Staubli VAL3: action_do.pgx

program action_do(ActionItem& x_aAction[] (dimensions=1), num x_nIndex (dimensions=1))
  local num i
  local num j
  local bool l_bExit
  local num l_nClock
  local num l_nDistance
  local num l_nResult
  local string l_sData
  local string l_sEmpty
  local string l_sInstr
  local string l_sInstruction
  local string l_sType
begin
  // check if not empty...
  if x_aAction.iInstr[0].sType!="" or x_aAction.iInstr[1].sType!="" or x_aAction.iInstr[2].sType!=""
    if saveData:bDebug
      ? "ACTION INSERT,"+x_aAction.iInstr.sType+" "+x_aAction.iInstr.sData+",ID="+toString(".3",getMoveId())+","+toString(".3",clock()-cycleStatus:nTime)+",x_ID="+toString("",x_aAction.nMoveId)+",x_Dist="+toString(".2",x_aAction.nDistance)
    endIf
    l_nClock=clock()
    // wait the correct moveID
    wait((x_aAction.nMoveId+x_aAction.nDistance)<=getMoveId() or (isEmpty()) and !cycleStatus:bPause)
    // look if there are several sAction in the traj
    for i=0 to (size(x_aAction.iInstr)-1)
      // check for not empty space
      if x_aAction.iInstr[i].sType!=""
        // get the instruction
        l_sData=x_aAction.iInstr[i].sData
        l_sType=x_aAction.iInstr[i].sType
        call saveInOut:replaceIO(l_sData,l_sType,l_sData)
        l_sInstr=l_sType+" "+l_sData
        if saveData:bDebug
          ? "ACTION RUNNING,"+l_sInstr+",ID="+toString(".3",getMoveId())+","+toString(".3",clock()-cycleStatus:nTime)+",MoveID="+toString("",x_aAction.nMoveId)+",Dist="+toString(".2",x_aAction.nDistance)
        endIf
        // PRINT LOG
        if cycleStatus:bCycle
          if x_aAction.nPointId!=-1
            // is inside a trajectory
            call cycleStatus:printLog(" ."+l_sInstr)
          else
            // is outside a trajectory
            call cycleStatus:printLog("-"+l_sInstr)
          endIf
        endIf
        cycleStatus:sToShow=l_sInstr
        cycleStatus:sLastAction=l_sInstr
        if x_aAction.nPointId==-1
          // refresh the LINE of the program...
          cycleStatus:bTraj=false
          cycleStatus:nEvent=x_nIndex
        endIf
        //
        // RUN THE ACTION
        //
        call memory_onRun(x_aAction.iInstr[i])
      endIf
    endFor
    // release
    cycleStatus:sToShow=""
  endIf
end
